{attribute 'GeneratedUsingTerminal: EL1008-0000-0018'}
{attribute addProperty BoxType "EL1008-0000-0018"}
{attribute addProperty Id "InputAT %I*BOOL1"}
{attribute addProperty CRC "2198356929"}
{attribute addProperty Size "1"}
TYPE Channel_830843C1 EXTENDS InputBase_8311D824 :
STRUCT
	{attribute addProperty Name "Input"}
	Input AT %I* : BOOL;
END_STRUCT
END_TYPE

(* stored: Version 1.2.0.0
   DUT Channel_830843C1: Id {b98ffb96-8777-4b28-8fa3-ef161d1a201c} *)
